// TwinCAT 3 PLC project HansPlc
// Title: Inxton
// Company: Inxton
// ProjectVersion: 0.0.0.1
// ProgramVersion: 3.1.4023.0
// libraries:
//   Tc2_Standard, * (Beckhoff Automation GmbH)
//   Tc2_System, * (Beckhoff Automation GmbH)
//   Tc3_Module, * (Beckhoff Automation GmbH)
// project tree:
//   Influx/ fbInfluxPerformanceLogging.TcPOU, InfluxData.TcDUT, prgInflux.TcPOU
//   / MAIN.TcPOU, PlcTask.TcTTO (not stored)
//   Mongo/ prgMongoDb.TcPOU, structMongoData.TcDUT
//   Recipes/ RecipeData.TcGVL, stContinuousValueLimits.TcDUT, stRecipe.TcDUT
//   VoiceSyntesis/ fbSpeech.TcPOU, prgVoiceSynsthesis.TcPOU
//   _Utils/ fbFluentString.TcPOU (not stored), fbSimpleRemoteExec.TcPOU (not stored), Utils.TcGVL (not stored)
//   WeatherStations/ enumStationStatus.TcDUT, fbWorldWeatherWatch.TcPOU, prgWeatherStations.TcPOU, structWeatherStation.TcDUT
// real-time tasks:
//   TASK PlcTask: cycle T#10ms, priority 20, ADS port 350

// ---- Influx/InfluxData.TcDUT
TYPE InfluxData :
STRUCT
	CycleCount : UDINT;
	CycleTime : UDINT;
	LastExecTime: UDINT;
	Minimum : UDINT := 0;
	Maximum : UDINT := 4294967295;	
END_STRUCT
END_TYPE

// ---- Mongo/structMongoData.TcDUT
TYPE structMongoData :
STRUCT
	CycleCount : UDINT;
	CycleTime : UDINT;
	LastExecTime: UDINT;
	Minimum : UDINT := 0;
	Maximum : UDINT := 4294967295;	
END_STRUCT
END_TYPE

// ---- Recipes/stContinuousValueLimits.TcDUT
{attribute wpf [Container(Layout.Wrap)]}
{attribute wpf [Group(Layout.GroupBox)]}
{attribute addProperty Name ""}
TYPE stContinuousValueLimits :
STRUCT	
	{attribute addProperty Name "<#Min#>"}
	Minimum : REAL;		
	{attribute addProperty Name "<#Acquired#>"}
	{attribute wpf [RenderIgnore("Control", "ShadowControl")]} // Prevents rednering this memember when 'PresentationType' is set to 'Control' or 'ShadowControl'.
	Acquired : REAL;	
	{attribute addProperty Name "<#Max#>"}
	Maximum : REAL;
END_STRUCT
END_TYPE

// ---- Recipes/stRecipe.TcDUT
TYPE stRecipe :
STRUCT
	{attribute addProperty Name "<#Recipe name#>"}
	_recipeName : STRING;
	{attribute addProperty Name "<#Description#>"}
	_description : STRING(255);
	// Uncomment following lines run the compiler and check that the fiels are added to the UI, and you can save and retrieve the newly added variables.
	{attribute addProperty Name "<#Length#> [mm]"}		
	_lenght : stContinuousValueLimits;	
	{attribute addProperty Name "<#Height#> [mm]"}
	_height : stContinuousValueLimits;
	{attribute addProperty Name "<#Thickness#> [mm]"}
	_thikness : stContinuousValueLimits;
END_STRUCT
END_TYPE

// ---- WeatherStations/enumStationStatus.TcDUT
{attribute 'qualified_only'}
{attribute 'strict'}
TYPE enumStationStatus :
(
	Unknown := 0,
	Available := 1,
	UnAvailable := 2	
);
END_TYPE

// ---- WeatherStations/structWeatherStation.TcDUT
{attribute wpf [Container(Layout.Stack)]}
{attribute addProperty OpenMap "https://www.openstreetmap.org/search?query=Kriva#map=13/49.2826/19.4791"}
TYPE structWeatherStation :
STRUCT
	{attribute addProperty Name "<#Station name (ICAO)#>"}	
	StationICAO : STRING(4);
	{attribute addProperty Name "<#Station status#>"}
    StationStatus : enumStationStatus; 
	{attribute addProperty Name "<#Dew Point#>"}	
	{attribute addProperty Units "°C"}
	DewPoint : REAL;
	{attribute addProperty Name "<#Pressure#>"}
    {attribute addProperty Units "Torr"}	
	Pressure : REAL;
	{attribute addProperty Name "<#Temperature#>"}
	{attribute addProperty Units "°C"}
	Temp : REAL;
	{attribute addProperty Name "<#Visibility#>"}
    {attribute addProperty Units "km"}	
	Visibility : REAL;			
	{attribute addProperty Name "<#Wind heading#>"}
    {attribute addProperty Units "Azimuth"}	
	WindHeading : UINT;	
	{attribute addProperty Name "<#Wind speed#>"}
    {attribute addProperty Units "m/s"}	
	WindSpeed : REAL;	
END_STRUCT
END_TYPE

// ---- Recipes/RecipeData.TcGVL
{attribute 'qualified_only'}
VAR_GLOBAL
	_recipe : stRecipe;
END_VAR

// ---- Influx/fbInfluxPerformanceLogging.TcPOU
FUNCTION_BLOCK fbInfluxPerformanceLogging
VAR
	{attribute clr [ReadOnly()]}
	{attribute clr [CompilerOmits("BuilderPlainer")]}
	{attribute clr [RenderIgnore()]}
	_logStart : ULINT;
	{attribute clr [RenderIgnore()]}
	{attribute clr [CompilerOmits("BuilderPlainer")]}
	_logDone : ULINT;
	
	_data : InfluxData;	
END_VAR

_data.CycleCount := TwinCAT_SystemInfoVarList._TaskInfo[1].CycleCount;
_data.CycleTime := TwinCAT_SystemInfoVarList._TaskInfo[1].CycleTime;
_data.LastExecTime := TwinCAT_SystemInfoVarList._TaskInfo[1].LastExecTime;

IF(_data.Maximum < _data.LastExecTime) THEN _data.Maximum := _data.LastExecTime; END_IF;
IF(_data.Minimum > _data.LastExecTime) THEN _data.Minimum := _data.LastExecTime; END_IF;

IF(_logStart <= _logDone) THEN 
	_logStart := _logStart + 1;	
END_IF

END_FUNCTION_BLOCK

// ---- Influx/prgInflux.TcPOU
PROGRAM prgInflux
VAR
	_influx : fbInfluxPerformanceLogging;
END_VAR

_influx();

END_PROGRAM

// ---- MAIN.TcPOU
PROGRAM MAIN

prgWeatherStations();
prgInflux();
prgMongoDb();

END_PROGRAM

// ---- WeatherStations/prgWeatherStations.TcPOU
{attribute addProperty Name "Program"}
{attribute wpf [Container(Layout.Stack)]}
PROGRAM prgWeatherStations
VAR	
	{attribute addProperty Name "Weather Cyclic"}
	_weatherStations : fbWorldWeatherWatch;	
	{attribute wpf [Container(Layout.Stack)]}
	{attribute wpf [Group(Layout.GroupBox)]}
    {attribute addProperty Name "<#What plc says#>"}	
	PlcCommentOnCurrentWeather : STRING(255) := 'TEST';	
END_VAR

_weatherStations();	
PlcCommentOnCurrentWeather := _weatherStations.PlcComments();

END_PROGRAM

// ---- WeatherStations/fbWorldWeatherWatch.TcPOU
{attribute wpf [Container(Layout.Tabs)]}
FUNCTION_BLOCK fbWorldWeatherWatch
VAR	
	{attribute addProperty Name "<#North pole station#>"}
	{attribute addProperty OpenMap "https://www.openstreetmap.org/?mlat=74.652&mlon=-95.556#map=6/74.652/-95.556"}
	NorthPole : structWeatherStation := (StationICAO := 'CYRB');
	{attribute addProperty Name "<#South pole station#>"}
	{attribute addProperty OpenMap "https://www.openstreetmap.org/?mlat=-85.05113&mlon=-16.80701#map=1/-85.05113/-16.80701"}
	SouthPole : structWeatherStation := (StationICAO := 'NZSP');
	{attribute addProperty Name "<#Verl, Germany#>"}
	{attribute addProperty OpenMap "https://www.openstreetmap.org/?mlat=51.5799&mlon=8.415#map=6/51.5799/8.4155"}
	Verl : structWeatherStation := (StationICAO := 'EDLP');
	{attribute addProperty Name "<#Kriva, Slovakia#>"}
	{attribute addProperty OpenMap "https://www.openstreetmap.org/?mlat=48.1723&mlon=17.2158#map=6/48.1723/17.2158"}
	Kriva : structWeatherStation := (StationICAO := 'LZIB');	
END_VAR

METHOD PlcComments : STRING[255]
VAR_INPUT
END_VAR
(* PLC IS COMMENTING ON WEATHER, GETTING INFORMATION FROM WEATHER STATIONS FROM ARROUND THE WORLD *)

Utils.FluentString.Append('<#So, the weather situation is following#>: $N');

IF (NorthPole.StationStatus = enumStationStatus.Available) THEN
	IF(NorthPole.Temp > -50) THEN
		Utils.FluentString.Append('<#It is fairly warm at the north pole.#>$N');
	ELSE
		Utils.FluentString.Append('<#It is as cold as it should be at the nort pole.#>$N');
	END_IF;
ELSE;
	Utils.FluentString.Append('<#North pole station is not available.#>$N');
END_IF; 


IF (SouthPole.StationStatus = enumStationStatus.Available) THEN
	IF(SouthPole.Temp > -50) THEN
		Utils.FluentString.Append('<#It is fairly warm at the south pole.#>$N');
	ELSE
		Utils.FluentString.Append('<#It is as cold as it should be at the souht pole.#>$N');
	END_IF; 
ELSE;
	Utils.FluentString.Append('<#South pole station is not available.#>$N');
END_IF; 


IF (Verl.StationStatus = enumStationStatus.Available) THEN
	IF(Verl.Temp > 0) THEN
		Utils.FluentString.Append('<#It is not freezing in Verl.#>$N');
	ELSE
		Utils.FluentString.Append('<#It is freezing in Verl.#>$N');
	END_IF; 
ELSE;
	Utils.FluentString.Append('<#Verl station is not available.#>$N');
END_IF; 


IF (Kriva.StationStatus = enumStationStatus.Available) THEN
	IF(Kriva.Temp > 0) THEN
		Utils.FluentString.Append('<#It is not freezing in Kriva.#>$N');
	ELSE
		Utils.FluentString.Append('<#It is freezing in Kriva.#>$N');
	END_IF; 
ELSE;
	Utils.FluentString.Append('<#Kriva station is not available.#>$N');
END_IF; 

PlcComments := Utils.FluentString.Result;
END_METHOD

END_FUNCTION_BLOCK

// ---- Mongo/prgMongoDb.TcPOU
PROGRAM prgMongoDb
VAR
	{attribute clr [ReadOnly()]}
	{attribute clr [CompilerOmits("BuilderPlainer")]}
	{attribute clr [RenderIgnore()]}
	_logStart : ULINT;
	{attribute clr [RenderIgnore()]}
	{attribute clr [CompilerOmits("BuilderPlainer")]}
	_logDone : ULINT;
	
	_data : structMongoData;
END_VAR

_data.CycleCount := TwinCAT_SystemInfoVarList._TaskInfo[1].CycleCount;
_data.CycleTime := TwinCAT_SystemInfoVarList._TaskInfo[1].CycleTime;
_data.LastExecTime := TwinCAT_SystemInfoVarList._TaskInfo[1].LastExecTime;

IF(_data.Maximum < _data.LastExecTime) THEN _data.Maximum := _data.LastExecTime; END_IF;
IF(_data.Minimum > _data.LastExecTime) THEN _data.Minimum := _data.LastExecTime; END_IF;

IF(_logStart <= _logDone) THEN 
	_logStart := _logStart + 1;	
END_IF

END_PROGRAM

// ---- VoiceSyntesis/fbSpeech.TcPOU
FUNCTION_BLOCK fbSpeech EXTENDS fbSimpleRemoteExec

METHOD  Execute : BOOL
VAR_INPUT
	param : ANY;
END_VAR
Speak(
END_METHOD

METHOD PRIVATE Speak : BOOL
VAR_INPUT
	_sentence : STRING(255);
END_VAR
END_METHOD

END_FUNCTION_BLOCK

// ---- VoiceSyntesis/prgVoiceSynsthesis.TcPOU
PROGRAM prgVoiceSynsthesis
VAR
END_VAR

END_PROGRAM
